// TIA Portal V20 export
DATA_BLOCK "IdentMvInterfaceHmi"   // DB219
// stored: InstanceOfName typeIdentMvHmi, InstanceOfType UDT
"typeIdentMvHmi"
   // VAR
   //    selectedUnit : USInt := 1;
   //    selectedEM : USInt := 6;
   //    mvReaderId : USInt := 0;
   //    numberOfMv : USInt := 1;
   //    mvReader : Array[0.."NO_OF_MV_IDENT_DEVICES"] of "LSicar_typeIdentInterfaceHmi";
   // END_VAR
BEGIN
   mvReader[0..1].deviceName := WSTRING#'';
   mvReader[0..1].deviceType := WSTRING#'';
   mvReader[0..1].deviceId := 0;
   mvReader[0..1].tagType := WSTRING#'';
   mvReader[0..1].cameraMode := WSTRING#'';
   mvReader[0..1].resultState := WSTRING#'';
   mvReader[0..1].progNo := 0;
   mvReader[0..1].progNumberWrite := 0;
   mvReader[0..1].pushbutton := 16#0000;
   mvReader[0..1].enablePushbutton := 16#0000;
   mvReader[0..1].status := 16#0000;
   mvReader[0..1].alarmCategorie := 0;
   mvReader[0..1].alarmNo := 0;
   mvReader[0..1].alarmCode := 16#0000_0000;
   mvReader[0..1].resultColor := 0;
   mvReader[0..1].statusColorCode := 0;
   mvReader[0..1].datRead1 := '';
   mvReader[0..1].datRead2 := '';
   mvReader[0..1].datRead3 := '';
   mvReader[0..1].datRead4 := '';
   mvReader[0..1].datWrite1 := '';
   mvReader[0..1].datWrite2 := '';
   mvReader[0..1].datWrite3 := '';
   mvReader[0..1].datWrite4 := '';
END_DATA_BLOCK
